TYPE ST_HMI :
STRUCT
	Inputs  : ST_Inputs;
	Status  : ST_ActuatorStatus;
	Config  : ST_ActuatorConfiguration;
	Fault   : ST_Error;
	
	OneShotClick : BOOL;
END_STRUCT
END_TYPE

(* stored: Version 1.1.0.1, ProductVersion 3.1.4024.12
   DUT ST_HMI: Id {08d8503e-6fe0-47bd-a1e3-0e667fd9ca36} *)
